FUNCTION_BLOCK FB_Unit
VAR
	step : (idle, init, Forward, Backward, Stop);
	Command : E_Command;
	fbTon : TON := (PT:=T#1S);
	bInit : BOOL;
	i : INT;
	
	
	(*Visu*)
	LED : ARRAY[1..10] OF BOOL;
	LEDLocation : ARRAY[1..2] OF INT;
	
	GenerateButton : FB_Button(E_Command.Generate);
	ForwardButton : FB_Button(E_Command.Forward);
	BackwardButton : FB_Button(E_Command.Backward);
	StopButton : FB_Button(E_Command.Stop);
END_VAR

IF NOT bInit THEN
	RETURN;
END_IF

IF Command = E_Command.Generate THEN
	LEDLocation[1] := 1;
	LEDLocation[2] := 2;
	step := Init;
	fbTon(IN := FALSE);
END_IF

CASE step OF
	Idle:
		;
	init:		
		fbTon(IN := TRUE);
		IF fbTon.Q THEN
			fbTon(IN := FALSE);
			IF Command = E_Command.Forward THEN
				step := Forward;
			ELSIF Command = E_Command.Backward THEN
				step := Backward;
			ELSIF Command = E_Command.Stop THEN
				step := Stop;
				fbTon(IN := FALSE);
			END_IF
		END_IF
	Forward:
		FOR i:= 1 TO 2 BY 1 DO
			IF LEDLocation[i] > 0 AND LEDLocation[i] <= 10 THEN
				LEDLocation[i] := LEDLocation[i] + 1;
			ELSE
				LEDLocation[i] := 0;
			END_IF 
		END_FOR
		fbTon(IN := TRUE);
		step := Init;
		
	Backward:
		FOR i:= 1 TO 2 BY 1 DO
			IF LEDLocation[i] > 0 AND LEDLocation[i] < 11 THEN
				LEDLocation[i] := LEDLocation[i] - 1;
			ELSE
				LEDLocation[i] := 0;
			END_IF 
		END_FOR
		fbTon(IN := TRUE);
		step := Init;
		
	Stop:
		IF Command = E_Command.Forward THEN
			fbTon(IN := TRUE);
			IF fbTon.Q THEN
				step := Forward;
				fbTon(IN := FALSE);
			END_IF
		ELSIF Command = E_Command.Backward THEN
			fbTon(IN := TRUE);
			IF fbTon.Q THEN
				step := Backward;
				fbTon(IN := FALSE);
			END_IF
		END_IF
END_CASE

TurnOnTwoLED(LEDLocation[1],LEDLocation[2]);
ForwardButton();
BackwardButton();
StopButton();
GenerateButton();

METHOD Initalize : BOOL
VAR_INPUT
	iLog : I_Log;
END_VAR
IF bInit THEN
	RETURN;
END_IF
ForwardButton.iLog := iLog;
ForwardButton.refCommand REF= Command;
BackwardButton.iLog := iLog;
BackwardButton.refCommand REF= Command;
StopButton.iLog := iLog;
StopButton.refCommand REF= Command;
GenerateButton.iLog := iLog;
GenerateButton.refCommand REF= Command;

bInit := TRUE;
END_METHOD

METHOD PRIVATE TurnOnTwoLED
VAR_INPUT
	Location1 : INT;
	Location2 : INT;
END_VAR
VAR
	i : INT;
END_VAR
IF Location1 = 0 AND Location2 = 0 THEN
	step := Idle;
END_IF

FOR i := 1 TO 10 BY 1 DO
	IF i = Location1 THEN
		LED[i] := TRUE;
	ELSIF i = Location2 THEN
		LED[i] := TRUE;
	ELSE
		LED[i] := FALSE;
	END_IF
END_FOR
END_METHOD

END_FUNCTION_BLOCK

(* stored: Version 1.1.0.1, ProductVersion 3.1.4024.12
   POU FB_Unit: Id {69683204-5b7b-42cd-b701-e61dc4d40a10}, SpecialFunc None
   Method Initalize: Id {86c290be-4fb0-45cd-a335-5538d682c0c9}
   Method TurnOnTwoLED: Id {b85f6523-b0b1-4239-8ed8-beb4292f26ee} *)
